# EPICS autosave request: iocBoot/iocCamera/ioc.req
file "camera.req",          P=$(P), R=cam1:
file "plugins.req",         P=$(P)
